(* Schneider Machine Expert - Basic project laba3, file version 2.5.0.0 *)
(* ProjectInformations: Name=New project *)

HARDWARE
  Cpu 0: TM221C16T
  Cartridge1 0: TMC2AQ2V
  EthernetConfiguration: NetworkName=M221, IpAllocationMode=FixedAddress, IpAddress=0.0.0.0, SubnetMask=0.0.0.0
  EthernetConfiguration: NetworkName=M221, IpAllocationMode=FixedAddress, IpAddress=0.0.0.0, SubnetMask=0.0.0.0
  SerialLineConfiguration: Baud=Baud19200, Parity=ParityEven, DataBits=DataBits8, StopBits=StopBits1, PhysicalMedium=PhysicalMediumRs485, TransmissionMode=TransmissionModeModbusRtu, SlaveId=1, Addressing=SlaveAddressing
  MastTask: UsePeriodScanMode=false, PeriodScan=100
  FastTask: Period=255
  CpuBehavior: StartingMode=StartAsPreviousState, AutoSaveRamOnEeprom=true, WatchdogPeriod=250

SYMBOLS  (address, symbol, comment, settings)
  %M10      SIM
  %M11      LS_LO_SIM
  %M12      LS_MID_SIM
  %M13      LS_HI_SIM
  %M100     S_IDLE
  %M101     S_LOAD1
  %M102     S_LOAD2
  %M103     S_HEA1
  %M104     S_HEA2
  %M105     S_DWNLD
  %M106     S_HOLD
  %S5       SB_TB100MS  "Time base of 100 ms generated by an internal clock"
  %S13      SB_FIRSTRUN  "Indicates the first controller cycle in RUN mode"
  %MW100    TE_SIM
  %MW101    LE_SIM
  %TM0        [Preset=30, Base=OneSecond]
  %I0.0     SB1_PUSK
  %I0.1     SB2_STOP
  %I0.2     LS1_LO
  %I0.3     LS2_MD
  %I0.4     LS3_HI
  %Q0.0     LVS1
  %Q0.1     LVS2
  %Q0.2     LVS3
  %IW0.0    TE1  [Type=Type_0_10V, Scope=Scope_Normal, Minimum=0, Maximum=1000]
  %QW0.100  TV1  [Type=Type_0_10V, Scope=Scope_Customized, Minimum=0, Maximum=10000]

POU New POU
  (* SectionNumber=1 *)

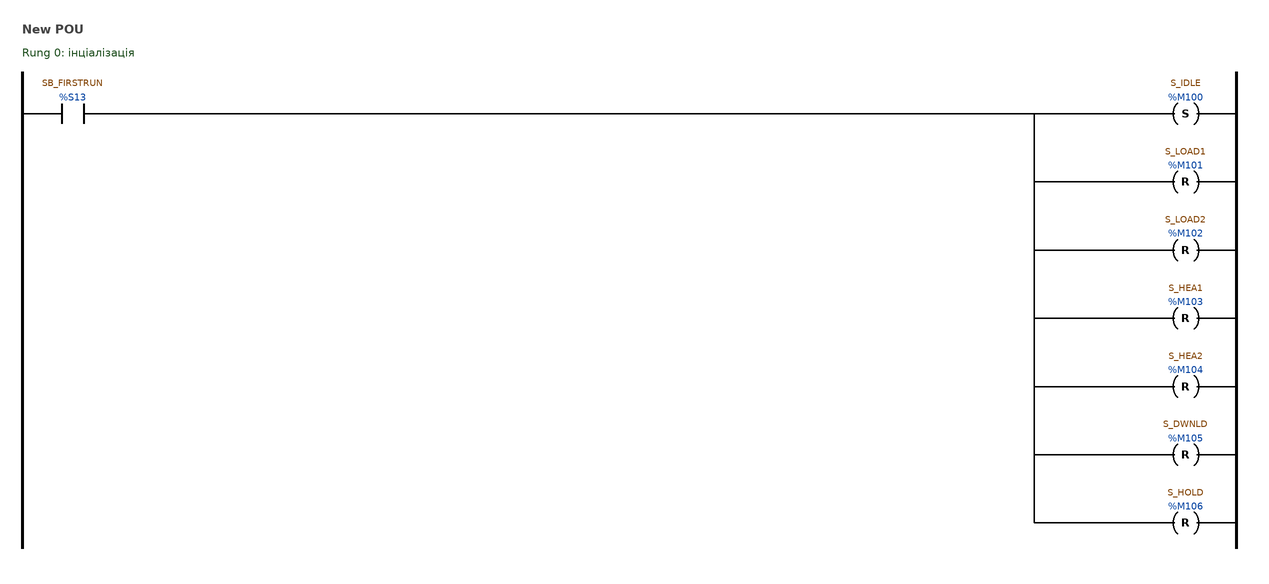

// Rung 0: інціалізація
  LD %S13                 (* SB_FIRSTRUN *)
  S %M100                 (* S_IDLE *)
  R %M101                 (* S_LOAD1 *)
  R %M102                 (* S_LOAD2 *)
  R %M103                 (* S_HEA1 *)
  R %M104                 (* S_HEA2 *)
  R %M105                 (* S_DWNLD *)
  R %M106                 (* S_HOLD *)
  // as ST:
  //   IF SB_FIRSTRUN THEN S_IDLE := TRUE; END_IF;
  //   IF SB_FIRSTRUN THEN S_LOAD1 := FALSE; END_IF;
  //   IF SB_FIRSTRUN THEN S_LOAD2 := FALSE; END_IF;
  //   IF SB_FIRSTRUN THEN S_HEA1 := FALSE; END_IF;
  //   IF SB_FIRSTRUN THEN S_HEA2 := FALSE; END_IF;
  //   IF SB_FIRSTRUN THEN S_DWNLD := FALSE; END_IF;
  //   IF SB_FIRSTRUN THEN S_HOLD := FALSE; END_IF;

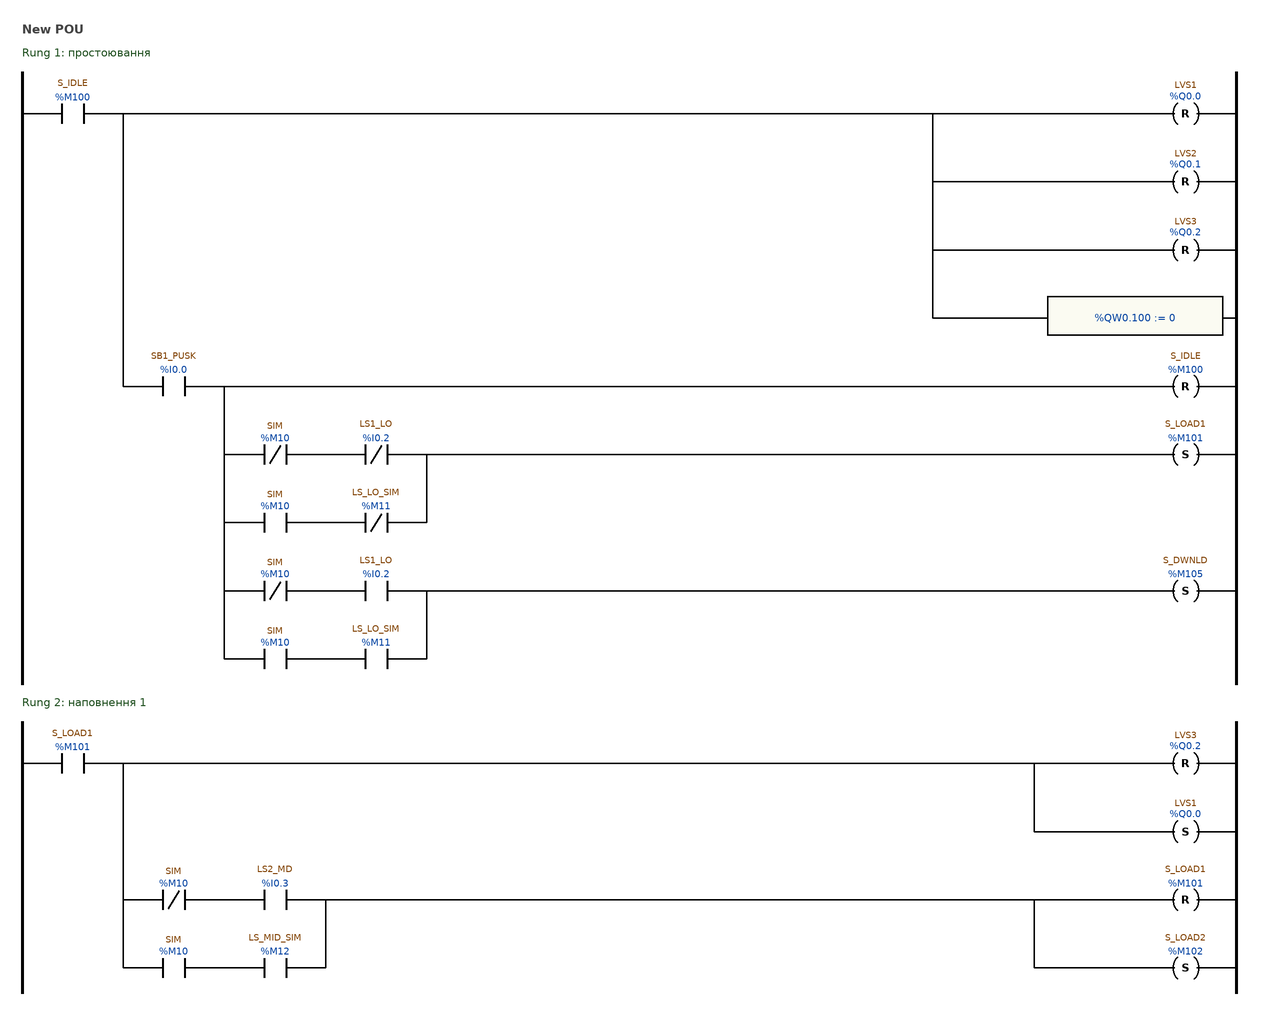

// Rung 1: простоювання
  LD %M100                (* S_IDLE *)
  MPS
  R %Q0.0                 (* LVS1 *)
  R %Q0.1                 (* LVS2 *)
  R %Q0.2                 (* LVS3 *)
  [ %QW0.100 := 0 ]       (* TV1 *)
  MPP
  AND %I0.0               (* SB1_PUSK *)
  MPS
  R %M100                 (* S_IDLE *)
  MRD
  AND(N %M10              (* SIM *)
  ANDN %I0.2              (* LS1_LO *)
  OR( %M10                (* SIM *)
  ANDN %M11               (* LS_LO_SIM *)
  )
  )
  S %M101                 (* S_LOAD1 *)
  MPP
  AND(N %M10              (* SIM *)
  AND %I0.2               (* LS1_LO *)
  OR( %M10                (* SIM *)
  AND %M11                (* LS_LO_SIM *)
  )
  )
  S %M105                 (* S_DWNLD *)
  // as ST:
  //   IF S_IDLE THEN LVS1 := FALSE; END_IF;
  //   IF S_IDLE THEN LVS2 := FALSE; END_IF;
  //   IF S_IDLE THEN LVS3 := FALSE; END_IF;
  //   IF S_IDLE THEN TV1 := 0; END_IF;
  //   _t1 := S_IDLE AND SB1_PUSK;
  //   IF _t1 THEN S_IDLE := FALSE; END_IF;
  //   IF _t1 AND (NOT SIM AND NOT LS1_LO OR SIM AND NOT LS_LO_SIM) THEN S_LOAD1 := TRUE; END_IF;
  //   IF _t1 AND (NOT SIM AND LS1_LO OR SIM AND LS_LO_SIM) THEN S_DWNLD := TRUE; END_IF;

// Rung 2: наповнення 1
  LD %M101                (* S_LOAD1 *)
  MPS
  R %Q0.2                 (* LVS3 *)
  S %Q0.0                 (* LVS1 *)
  MPP
  AND(N %M10              (* SIM *)
  AND %I0.3               (* LS2_MD *)
  OR( %M10                (* SIM *)
  AND %M12                (* LS_MID_SIM *)
  )
  )
  R %M101                 (* S_LOAD1 *)
  S %M102                 (* S_LOAD2 *)
  // as ST:
  //   IF S_LOAD1 THEN LVS3 := FALSE; END_IF;
  //   IF S_LOAD1 THEN LVS1 := TRUE; END_IF;
  //   _t1 := S_LOAD1 AND (NOT SIM AND LS2_MD OR SIM AND LS_MID_SIM);
  //   IF _t1 THEN S_LOAD1 := FALSE; END_IF;
  //   IF _t1 THEN S_LOAD2 := TRUE; END_IF;

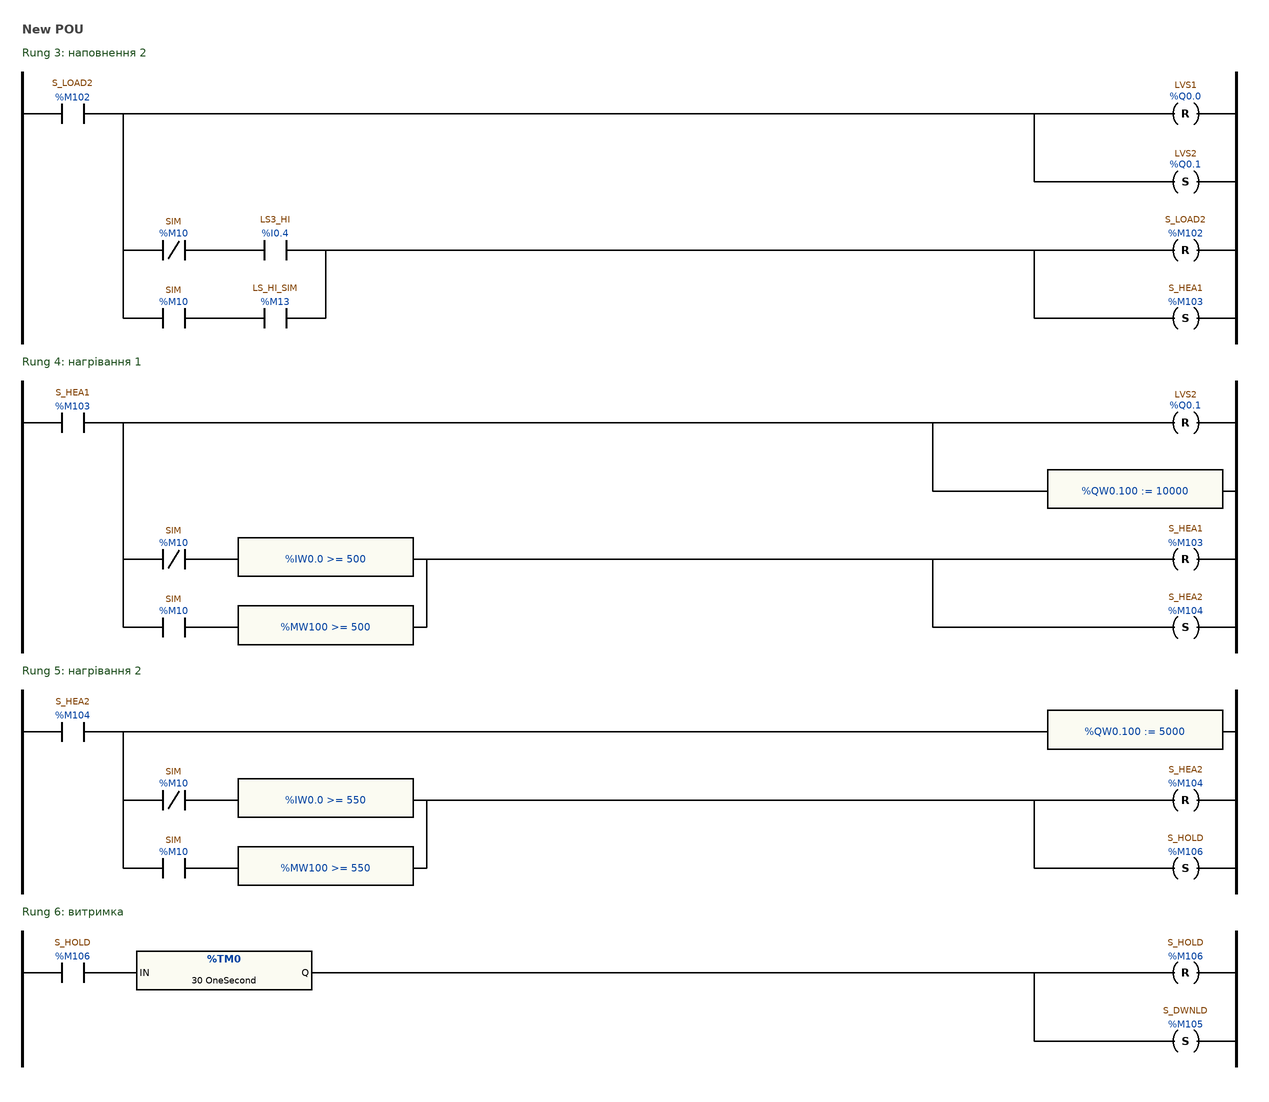

// Rung 3: наповнення 2
  LD %M102                (* S_LOAD2 *)
  MPS
  R %Q0.0                 (* LVS1 *)
  S %Q0.1                 (* LVS2 *)
  MPP
  AND(N %M10              (* SIM *)
  AND %I0.4               (* LS3_HI *)
  OR( %M10                (* SIM *)
  AND %M13                (* LS_HI_SIM *)
  )
  )
  R %M102                 (* S_LOAD2 *)
  S %M103                 (* S_HEA1 *)
  // as ST:
  //   IF S_LOAD2 THEN LVS1 := FALSE; END_IF;
  //   IF S_LOAD2 THEN LVS2 := TRUE; END_IF;
  //   _t1 := S_LOAD2 AND (NOT SIM AND LS3_HI OR SIM AND LS_HI_SIM);
  //   IF _t1 THEN S_LOAD2 := FALSE; END_IF;
  //   IF _t1 THEN S_HEA1 := TRUE; END_IF;

// Rung 4: нагрівання 1
  LD %M103                (* S_HEA1 *)
  MPS
  R %Q0.1                 (* LVS2 *)
  [ %QW0.100 := 10000 ]   (* TV1 *)
  MPP
  AND(N %M10              (* SIM *)
  AND [ %IW0.0 >= 500 ]   (* TE1 *)
  OR( %M10                (* SIM *)
  AND [ %MW100 >= 500 ]   (* TE_SIM *)
  )
  )
  R %M103                 (* S_HEA1 *)
  S %M104                 (* S_HEA2 *)
  // as ST:
  //   IF S_HEA1 THEN LVS2 := FALSE; END_IF;
  //   IF S_HEA1 THEN TV1 := 10000; END_IF;
  //   _t1 := S_HEA1 AND (NOT SIM AND TE1 >= 500 OR SIM AND TE_SIM >= 500);
  //   IF _t1 THEN S_HEA1 := FALSE; END_IF;
  //   IF _t1 THEN S_HEA2 := TRUE; END_IF;

// Rung 5: нагрівання 2
  LD %M104                (* S_HEA2 *)
  MPS
  [ %QW0.100 := 5000 ]    (* TV1 *)
  MPP
  AND(N %M10              (* SIM *)
  AND [ %IW0.0 >= 550 ]   (* TE1 *)
  OR( %M10                (* SIM *)
  AND [ %MW100 >= 550 ]   (* TE_SIM *)
  )
  )
  R %M104                 (* S_HEA2 *)
  S %M106                 (* S_HOLD *)
  // as ST:
  //   IF S_HEA2 THEN TV1 := 5000; END_IF;
  //   _t1 := S_HEA2 AND (NOT SIM AND TE1 >= 550 OR SIM AND TE_SIM >= 550);
  //   IF _t1 THEN S_HEA2 := FALSE; END_IF;
  //   IF _t1 THEN S_HOLD := TRUE; END_IF;

// Rung 6: витримка
  BLK %TM0
  LD %M106                (* S_HOLD *)
  IN
  OUT_BLK
  LD Q
  R %M106                 (* S_HOLD *)
  S %M105                 (* S_DWNLD *)
  END_BLK
  // as ST:
  //   %TM0(IN := S_HOLD);
  //   IF %TM0.Q THEN S_HOLD := FALSE; END_IF;
  //   IF %TM0.Q THEN S_DWNLD := TRUE; END_IF;

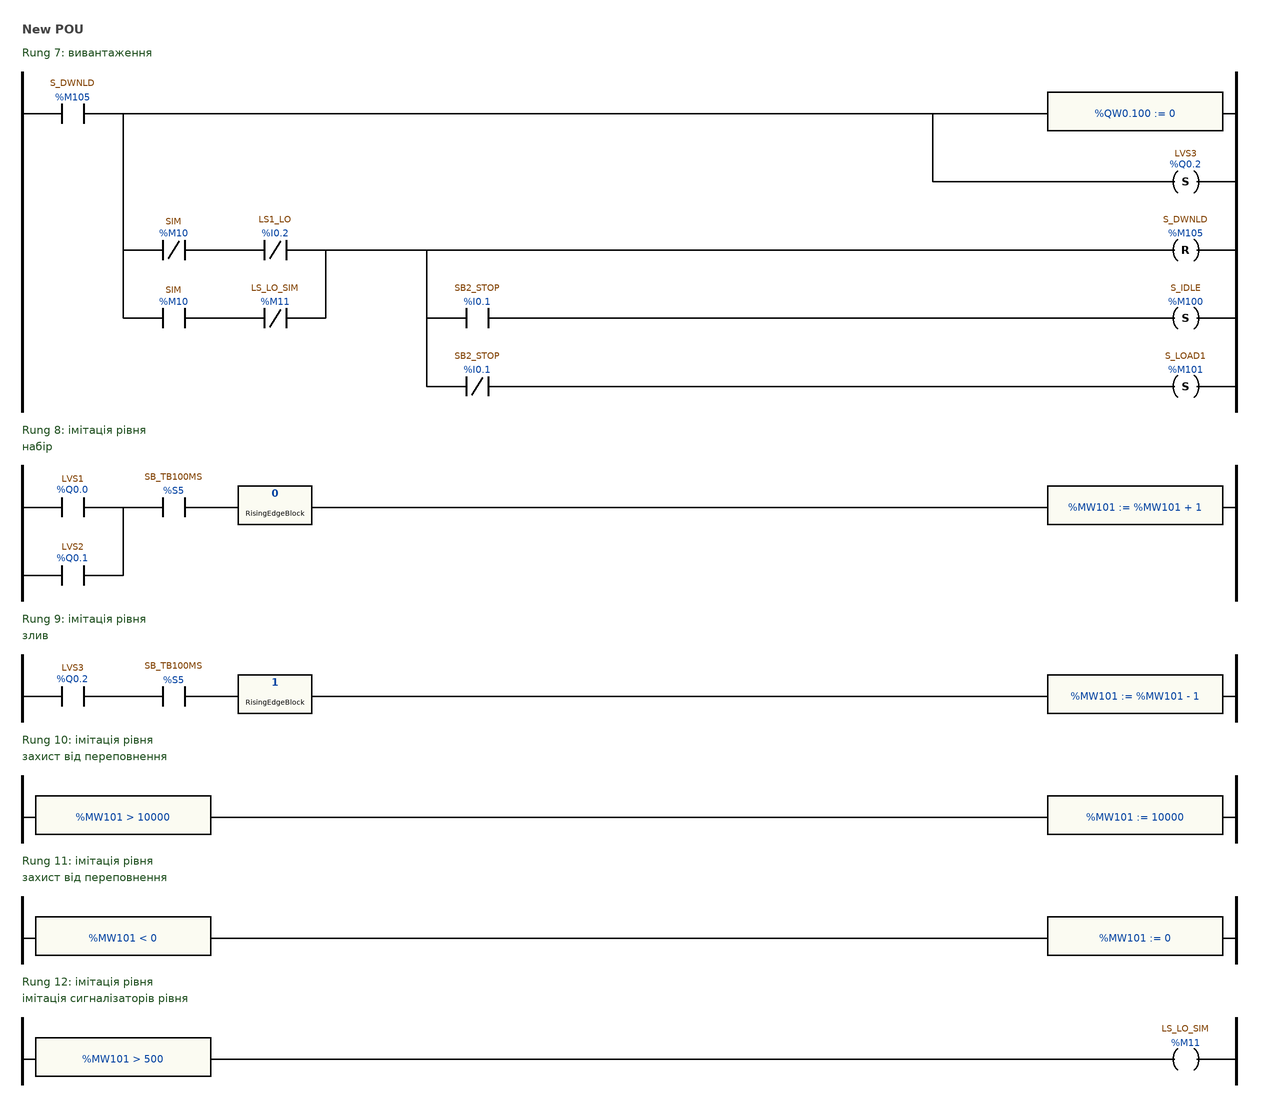

// Rung 7: вивантаження
  LD %M105                (* S_DWNLD *)
  MPS
  [ %QW0.100 := 0 ]       (* TV1 *)
  S %Q0.2                 (* LVS3 *)
  MPP
  AND(N %M10              (* SIM *)
  ANDN %I0.2              (* LS1_LO *)
  OR( %M10                (* SIM *)
  ANDN %M11               (* LS_LO_SIM *)
  )
  )
  MPS
  R %M105                 (* S_DWNLD *)
  MRD
  AND %I0.1               (* SB2_STOP *)
  S %M100                 (* S_IDLE *)
  MPP
  ANDN %I0.1              (* SB2_STOP *)
  S %M101                 (* S_LOAD1 *)
  // as ST:
  //   IF S_DWNLD THEN TV1 := 0; END_IF;
  //   IF S_DWNLD THEN LVS3 := TRUE; END_IF;
  //   _t1 := S_DWNLD AND (NOT SIM AND NOT LS1_LO OR SIM AND NOT LS_LO_SIM);
  //   IF _t1 THEN S_DWNLD := FALSE; END_IF;
  //   IF _t1 AND SB2_STOP THEN S_IDLE := TRUE; END_IF;
  //   IF _t1 AND NOT SB2_STOP THEN S_LOAD1 := TRUE; END_IF;

// Rung 8: імітація рівня
// набір
  LD %Q0.0                (* LVS1 *)
  OR %Q0.1                (* LVS2 *)
  AND %S5                 (* SB_TB100MS *)
  RISING0
  [ %MW101 := %MW101 + 1 ](* LE_SIM, LE_SIM *)
  // as ST:
  //   IF RISING((LVS1 OR LVS2) AND SB_TB100MS) THEN LE_SIM := LE_SIM + 1; END_IF;

// Rung 9: імітація рівня
// злив
  LD %Q0.2                (* LVS3 *)
  AND %S5                 (* SB_TB100MS *)
  RISING1
  [ %MW101 := %MW101 - 1 ](* LE_SIM, LE_SIM *)
  // as ST:
  //   IF RISING(LVS3 AND SB_TB100MS) THEN LE_SIM := LE_SIM - 1; END_IF;

// Rung 10: імітація рівня
// захист від переповнення
  LD [ %MW101 > 10000 ]   (* LE_SIM *)
  [ %MW101 := 10000 ]     (* LE_SIM *)
  // as ST:
  //   IF LE_SIM > 10000 THEN LE_SIM := 10000; END_IF;

// Rung 11: імітація рівня
// захист від переповнення
  LD [ %MW101 < 0 ]       (* LE_SIM *)
  [ %MW101 := 0 ]         (* LE_SIM *)
  // as ST:
  //   IF LE_SIM < 0 THEN LE_SIM := 0; END_IF;

// Rung 12: імітація рівня
// імітація сигналізаторів рівня
  LD [ %MW101 > 500 ]     (* LE_SIM *)
  ST %M11                 (* LS_LO_SIM *)
  // as ST:
  //   LS_LO_SIM := LE_SIM > 500;

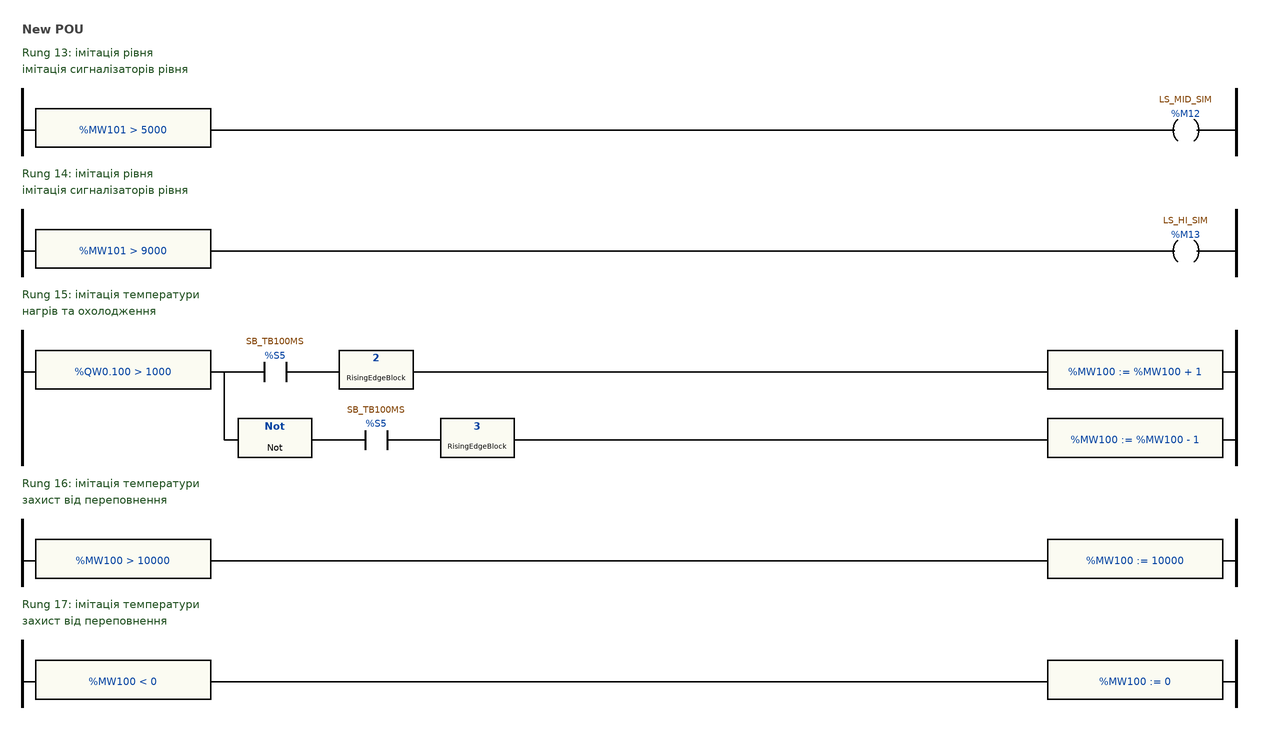

// Rung 13: імітація рівня
// імітація сигналізаторів рівня
  LD [ %MW101 > 5000 ]    (* LE_SIM *)
  ST %M12                 (* LS_MID_SIM *)
  // as ST:
  //   LS_MID_SIM := LE_SIM > 5000;

// Rung 14: імітація рівня
// імітація сигналізаторів рівня
  LD [ %MW101 > 9000 ]    (* LE_SIM *)
  ST %M13                 (* LS_HI_SIM *)
  // as ST:
  //   LS_HI_SIM := LE_SIM > 9000;

// Rung 15: імітація температури
// нагрів та охолодження
  LD [ %QW0.100 > 1000 ]  (* TV1 *)
  MPS
  AND %S5                 (* SB_TB100MS *)
  RISING2
  [ %MW100 := %MW100 + 1 ](* TE_SIM, TE_SIM *)
  MPP
  N
  AND %S5                 (* SB_TB100MS *)
  RISING3
  [ %MW100 := %MW100 - 1 ](* TE_SIM, TE_SIM *)
  // as ST:
  //   IF RISING(TV1 > 1000 AND SB_TB100MS) THEN TE_SIM := TE_SIM + 1; END_IF;
  //   IF RISING(NOT (TV1 > 1000) AND SB_TB100MS) THEN TE_SIM := TE_SIM - 1; END_IF;

// Rung 16: імітація температури
// захист від переповнення
  LD [ %MW100 > 10000 ]   (* TE_SIM *)
  [ %MW100 := 10000 ]     (* TE_SIM *)
  // as ST:
  //   IF TE_SIM > 10000 THEN TE_SIM := 10000; END_IF;

// Rung 17: імітація температури
// захист від переповнення
  LD [ %MW100 < 0 ]       (* TE_SIM *)
  [ %MW100 := 0 ]         (* TE_SIM *)
  // as ST:
  //   IF TE_SIM < 0 THEN TE_SIM := 0; END_IF;
